KUKA KRL data list: BaseCalib.dat

&ACCESS RV
DEFDAT BaseCalib PUBLIC

ENDDAT
